{attribute 'linkalways'} 
{attribute 'no_explicit_call' := 'This FB is a CLASS and must be accessed using methods or properties'}
{attribute 'enable_dynamic_creation'}
FUNCTION_BLOCK ABSTRACT MiddlewareBase implements I_Middleware
VAR
	_next : I_Middleware;
END_VAR

METHOD PUBLIC ABSTRACT Handle
VAR_INPUT
	Request : I_Request;
	Response : I_ServerResponse;
END_VAR
// Call next to pass the request and response to the next handler
// Next(Request, Response);
END_METHOD

METHOD PROTECTED Next
VAR_INPUT
	Request : I_Request;
	Response : I_ServerResponse;
END_VAR
IF _next = 0 THEN
	RETURN;
END_IF

_next.Handle(Request, Response);
END_METHOD

PROPERTY PUBLIC NextMiddleware : I_Middleware
GET
NextMiddleware := _next;
END_GET
SET
_next := NextMiddleware;
END_SET
END_PROPERTY

END_FUNCTION_BLOCK

(* stored: Version 1.1.0.1, ProductVersion 3.1.4026.13
   POU MiddlewareBase: Id {6733d455-3552-492f-84de-b78867d11567}, SpecialFunc None
   Folder Protected: Id {86f97faa-3f8f-469d-ba8e-49f9786f49da}
   Method Handle: Id {824c41b9-6692-4bc2-adbe-84668551a7c2}
   Method Next: Id {4e7f5e7b-0dbc-4379-8fce-ee24a6e2cbab}
   Property NextMiddleware: Id {672894c2-cba5-45a0-9770-82a8e8470631}
   Get Get: Id {da3262cc-76df-47ef-9585-d091cb913f14}
   Set Set: Id {9adafe75-c110-453f-a98a-cf262df9c2dd} *)
